// TIA Portal V21 export
VAR_GLOBAL   // PLC tag table "Tabella delle variabili standard"
   Tag_1 AT %M1.0 : Bool;
   "ALWAYS OFF" AT %M1.7 : Bool;
   Tag_2 AT %M21.0 : Bool;
   Tag_3 AT %T1000 : Timer;
   Tag_4 AT %MB22 : Byte;
   Tag_5 AT %M21.2 : Bool;
END_VAR
